TYPE "bwu4067CustomOutput16bytes"
TITLE = {"version":"v1.0","author":"cyanezf","family":"core/controller/bihl-wiedermann/bwu4067","status":"current","deprecatedBy": null,"dependencies":[]}

//(*--
//# Documentation
//## Log
//| version | date | author | description |
//|:-------:|:----:|:------:|:------------|
//| v1.0 | 2025-03-03 | cyanezf | First version |
//
//## Description
//B+W - bwu4067 Custom Output 16 bytes
//--*)

   STRUCT
      p1_spare : DWord;   // Reserved Io-link port
      p2_encoder : Struct   // BW4067-16bytes/Port 2-4bytes: Encoder
         dword1 : DWord;
         dword2 : DWord;
      END_STRUCT;
      p3_distance : DWord;   // BW4067-16bytes/Port 3-4bytes: Distance sensor
      p4_distance : DWord;   // BW4067-16bytes/Port 4-4bytes: Distance sensor
      spare : DWord;   // Free bytes
   END_STRUCT;

END_TYPE
